// TIA Portal V19 export
FUNCTION "MGF AUTO" : Void   // FC10, LAD
{ S7_Optimized_Access := 'TRUE' }
// stored: SetENOAutomatically false
BEGIN

REGION Network 1
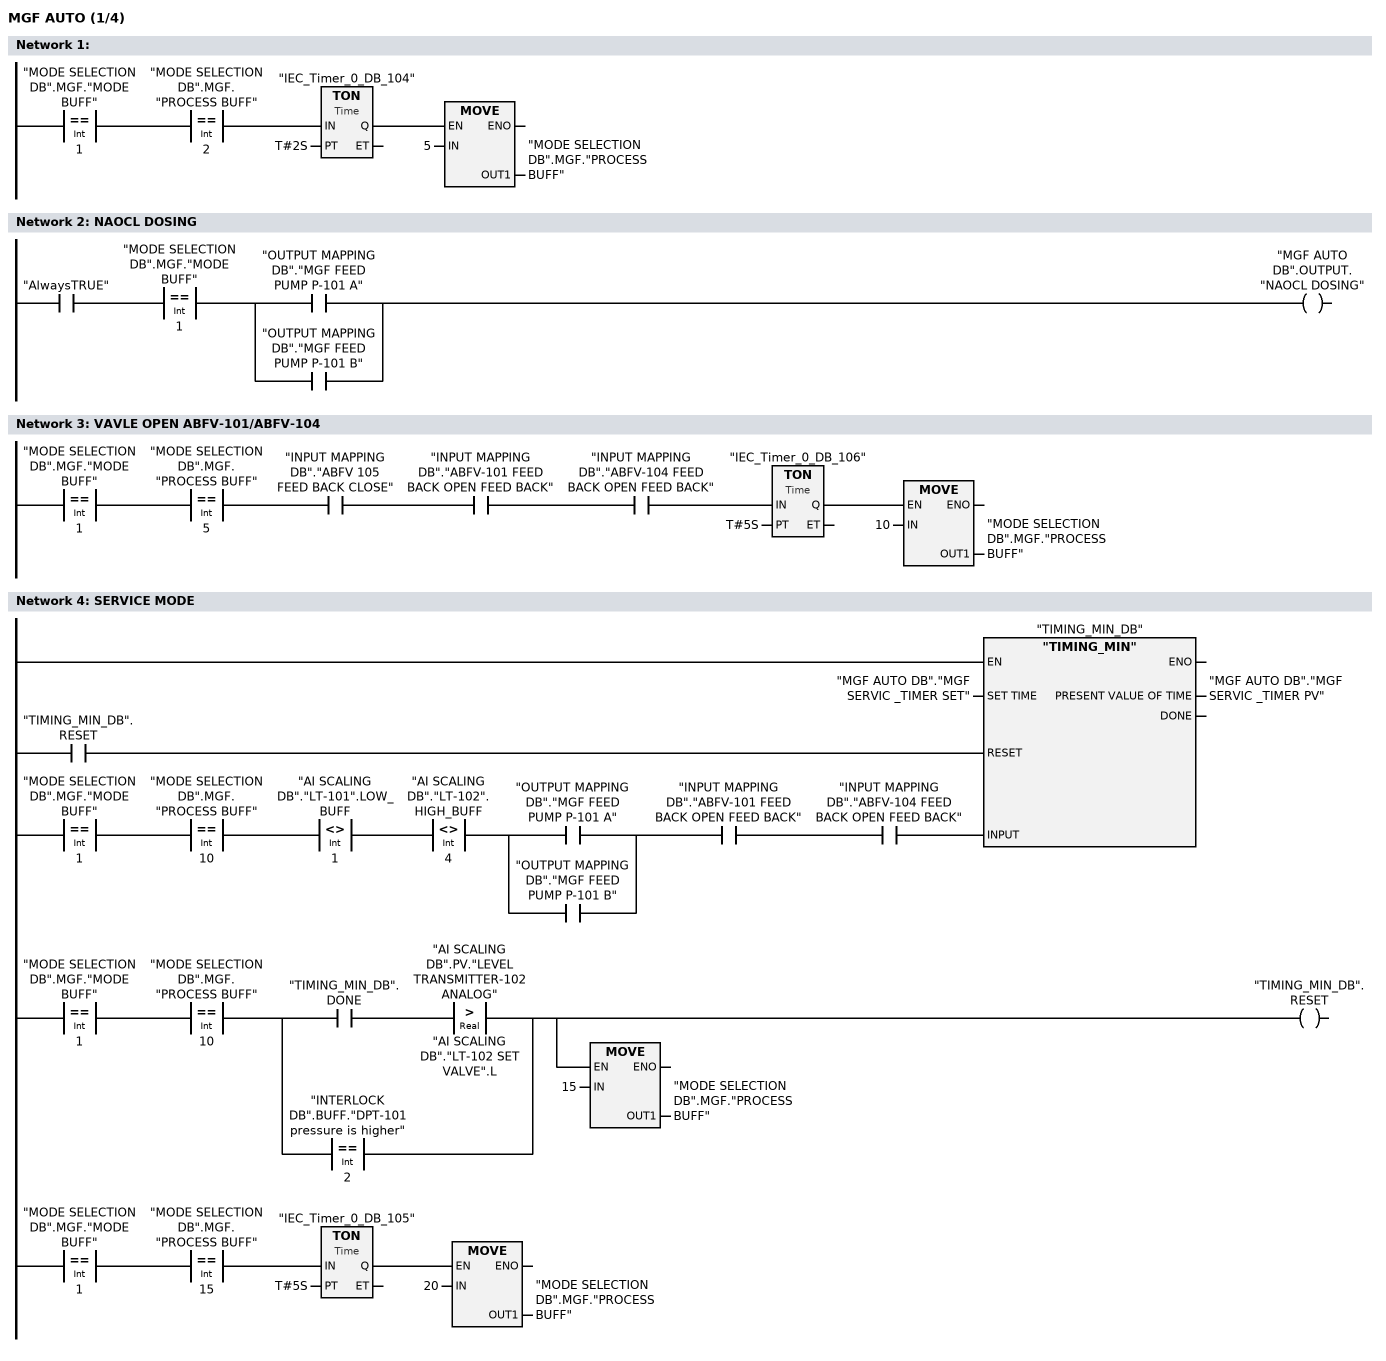
   RUNG wire#powerrail
      { S7_Templates := "SrcType := Int" } EQ_Contact(in1 := "MODE SELECTION DB".MGF."MODE BUFF", in2 := 1)
      { S7_Templates := "SrcType := Int" } EQ_Contact(in1 := "MODE SELECTION DB".MGF."PROCESS BUFF", in2 := 2)
      { S7_Templates := "time_type := Time" } "IEC_Timer_0_DB_104".TON(pt := T#2S, et =>)
      Move(in := 5, out1 => "MODE SELECTION DB".MGF."PROCESS BUFF")
   END_RUNG
   // the same network as SCL:
   "IEC_Timer_0_DB_104".TON(IN := ("MODE SELECTION DB".MGF."MODE BUFF" = 1) AND ("MODE SELECTION DB".MGF."PROCESS BUFF" = 2),
                           PT := T#2S);
   IF "IEC_Timer_0_DB_104".Q THEN "MODE SELECTION DB".MGF."PROCESS BUFF" := 5; END_IF;
END_REGION

REGION Network 2: NAOCL DOSING
   RUNG wire#powerrail
      Contact( "AlwaysTRUE" )
      { S7_Templates := "SrcType := Int" } EQ_Contact(in1 := "MODE SELECTION DB".MGF."MODE BUFF", in2 := 1)
      wire#w1
      Contact( "OUTPUT MAPPING DB"."MGF FEED PUMP P-101 A" )
      wire#w2
      Coil( "MGF AUTO DB".OUTPUT."NAOCL DOSING" )
   END_RUNG
   RUNG wire#w1
      Contact( "OUTPUT MAPPING DB"."MGF FEED PUMP P-101 B" )
   END_RUNG wire#w2
   // the same network as SCL:
   "MGF AUTO DB".OUTPUT."NAOCL DOSING" := "AlwaysTRUE" AND ("MODE SELECTION DB".MGF."MODE BUFF" = 1) AND ("OUTPUT MAPPING DB"."MGF FEED PUMP P-101 A" OR "OUTPUT MAPPING DB"."MGF FEED PUMP P-101 B");
END_REGION

REGION Network 3: VAVLE OPEN ABFV-101/ABFV-104
   RUNG wire#powerrail
      { S7_Templates := "SrcType := Int" } EQ_Contact(in1 := "MODE SELECTION DB".MGF."MODE BUFF", in2 := 1)
      { S7_Templates := "SrcType := Int" } EQ_Contact(in1 := "MODE SELECTION DB".MGF."PROCESS BUFF", in2 := 5)
      Contact( "INPUT MAPPING DB"."ABFV 105 FEED BACK CLOSE" )
      Contact( "INPUT MAPPING DB"."ABFV-101 FEED BACK OPEN FEED BACK" )
      Contact( "INPUT MAPPING DB"."ABFV-104 FEED BACK OPEN FEED BACK" )
      { S7_Templates := "time_type := Time" } "IEC_Timer_0_DB_106".TON(pt := T#5S, et =>)
      Move(in := 10, out1 => "MODE SELECTION DB".MGF."PROCESS BUFF")
   END_RUNG
   // the same network as SCL:
   "IEC_Timer_0_DB_106".TON(IN := ("MODE SELECTION DB".MGF."MODE BUFF" = 1) AND ("MODE SELECTION DB".MGF."PROCESS BUFF" = 5) AND "INPUT MAPPING DB"."ABFV 105 FEED BACK CLOSE" AND "INPUT MAPPING DB"."ABFV-101 FEED BACK OPEN FEED BACK" AND "INPUT MAPPING DB"."ABFV-104 FEED BACK OPEN FEED BACK",
                           PT := T#5S);
   IF "IEC_Timer_0_DB_106".Q THEN "MODE SELECTION DB".MGF."PROCESS BUFF" := 10; END_IF;
END_REGION

REGION Network 4: SERVICE MODE
   RUNG wire#powerrail
      "TIMING_MIN_DB"(RESET := wire#w1, INPUT := wire#w4, "SET TIME" := "MGF AUTO DB"."MGF SERVIC _TIMER SET", "PRESENT VALUE OF TIME" => "MGF AUTO DB"."MGF SERVIC _TIMER PV", DONE =>)
   END_RUNG
   RUNG wire#powerrail
      Contact( "TIMING_MIN_DB".RESET )
   END_RUNG wire#w1
   RUNG wire#powerrail
      { S7_Templates := "SrcType := Int" } EQ_Contact(in1 := "MODE SELECTION DB".MGF."MODE BUFF", in2 := 1)
      { S7_Templates := "SrcType := Int" } EQ_Contact(in1 := "MODE SELECTION DB".MGF."PROCESS BUFF", in2 := 10)
      { S7_Templates := "SrcType := Int" } NE_Contact(in1 := "AI SCALING DB"."LT-101".LOW_BUFF, in2 := 1)
      { S7_Templates := "SrcType := Int" } NE_Contact(in1 := "AI SCALING DB"."LT-102".HIGH_BUFF, in2 := 4)
      wire#w2
      Contact( "OUTPUT MAPPING DB"."MGF FEED PUMP P-101 A" )
      wire#w3
      Contact( "INPUT MAPPING DB"."ABFV-101 FEED BACK OPEN FEED BACK" )
      Contact( "INPUT MAPPING DB"."ABFV-104 FEED BACK OPEN FEED BACK" )
   END_RUNG wire#w4
   RUNG wire#w2
      Contact( "OUTPUT MAPPING DB"."MGF FEED PUMP P-101 B" )
   END_RUNG wire#w3
   RUNG wire#powerrail
      { S7_Templates := "SrcType := Int" } EQ_Contact(in1 := "MODE SELECTION DB".MGF."MODE BUFF", in2 := 1)
      { S7_Templates := "SrcType := Int" } EQ_Contact(in1 := "MODE SELECTION DB".MGF."PROCESS BUFF", in2 := 10)
      wire#w5
      Contact( "TIMING_MIN_DB".DONE )
      { S7_Templates := "SrcType := Real" } GT_Contact(in1 := "AI SCALING DB".PV."LEVEL TRANSMITTER-102 ANALOG", in2 := "AI SCALING DB"."LT-102 SET VALVE".L)
      wire#w6
      Coil( "TIMING_MIN_DB".RESET )
   END_RUNG
   RUNG wire#w5
      { S7_Templates := "SrcType := Int" } EQ_Contact(in1 := "INTERLOCK DB".BUFF."DPT-101 pressure is higher", in2 := 2)
   END_RUNG wire#w6
   RUNG wire#w6
      Move(in := 15, out1 => "MODE SELECTION DB".MGF."PROCESS BUFF")
   END_RUNG
   RUNG wire#powerrail
      { S7_Templates := "SrcType := Int" } EQ_Contact(in1 := "MODE SELECTION DB".MGF."MODE BUFF", in2 := 1)
      { S7_Templates := "SrcType := Int" } EQ_Contact(in1 := "MODE SELECTION DB".MGF."PROCESS BUFF", in2 := 15)
      { S7_Templates := "time_type := Time" } "IEC_Timer_0_DB_105".TON(pt := T#5S, et =>)
      Move(in := 20, out1 => "MODE SELECTION DB".MGF."PROCESS BUFF")
   END_RUNG
   // the same network as SCL:
   "TIMING_MIN_DB"("SET TIME" := "MGF AUTO DB"."MGF SERVIC _TIMER SET",   // "TIMING_MIN"
                   RESET := "TIMING_MIN_DB".RESET,
                   INPUT := ("MODE SELECTION DB".MGF."MODE BUFF" = 1) AND ("MODE SELECTION DB".MGF."PROCESS BUFF" = 10) AND ("AI SCALING DB"."LT-101".LOW_BUFF <> 1) AND ("AI SCALING DB"."LT-102".HIGH_BUFF <> 4) AND ("OUTPUT MAPPING DB"."MGF FEED PUMP P-101 A" OR "OUTPUT MAPPING DB"."MGF FEED PUMP P-101 B") AND "INPUT MAPPING DB"."ABFV-101 FEED BACK OPEN FEED BACK" AND "INPUT MAPPING DB"."ABFV-104 FEED BACK OPEN FEED BACK",
                   "PRESENT VALUE OF TIME" => "MGF AUTO DB"."MGF SERVIC _TIMER PV");
   "TIMING_MIN_DB".RESET := ("MODE SELECTION DB".MGF."MODE BUFF" = 1) AND ("MODE SELECTION DB".MGF."PROCESS BUFF" = 10) AND (("TIMING_MIN_DB".DONE AND ("AI SCALING DB".PV."LEVEL TRANSMITTER-102 ANALOG" > "AI SCALING DB"."LT-102 SET VALVE".L)) OR ("INTERLOCK DB".BUFF."DPT-101 pressure is higher" = 2));
   IF "TIMING_MIN_DB".RESET THEN "MODE SELECTION DB".MGF."PROCESS BUFF" := 15; END_IF;
   "IEC_Timer_0_DB_105".TON(IN := ("MODE SELECTION DB".MGF."MODE BUFF" = 1) AND ("MODE SELECTION DB".MGF."PROCESS BUFF" = 15),
                           PT := T#5S);
   IF "IEC_Timer_0_DB_105".Q THEN "MODE SELECTION DB".MGF."PROCESS BUFF" := 20; END_IF;
END_REGION

REGION Network 5: VAVLE CLOSE ABFV-101/ABFV-104
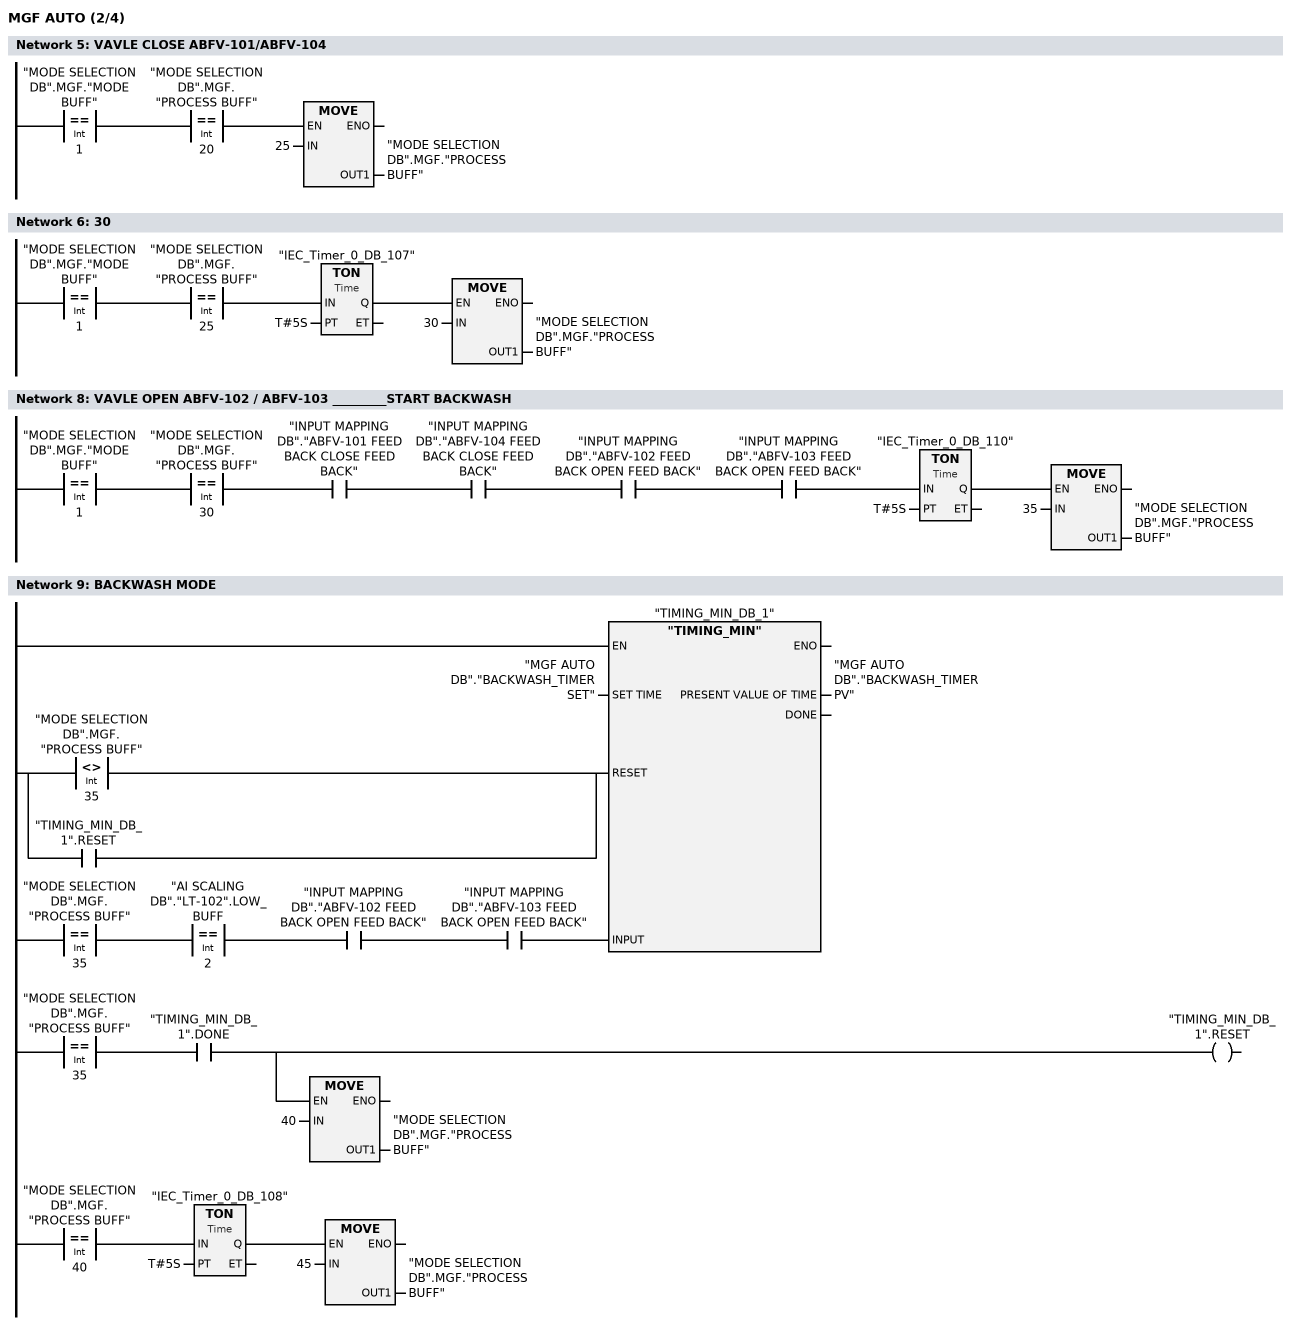
   RUNG wire#powerrail
      { S7_Templates := "SrcType := Int" } EQ_Contact(in1 := "MODE SELECTION DB".MGF."MODE BUFF", in2 := 1)
      { S7_Templates := "SrcType := Int" } EQ_Contact(in1 := "MODE SELECTION DB".MGF."PROCESS BUFF", in2 := 20)
      Move(in := 25, out1 => "MODE SELECTION DB".MGF."PROCESS BUFF")
   END_RUNG
   // the same network as SCL:
   IF ("MODE SELECTION DB".MGF."MODE BUFF" = 1) AND ("MODE SELECTION DB".MGF."PROCESS BUFF" = 20) THEN
       "MODE SELECTION DB".MGF."PROCESS BUFF" := 25;
   END_IF;
END_REGION

REGION Network 6: 30
   RUNG wire#powerrail
      { S7_Templates := "SrcType := Int" } EQ_Contact(in1 := "MODE SELECTION DB".MGF."MODE BUFF", in2 := 1)
      { S7_Templates := "SrcType := Int" } EQ_Contact(in1 := "MODE SELECTION DB".MGF."PROCESS BUFF", in2 := 25)
      { S7_Templates := "time_type := Time" } "IEC_Timer_0_DB_107".TON(pt := T#5S, et =>)
      Move(in := 30, out1 => "MODE SELECTION DB".MGF."PROCESS BUFF")
   END_RUNG
   // the same network as SCL:
   "IEC_Timer_0_DB_107".TON(IN := ("MODE SELECTION DB".MGF."MODE BUFF" = 1) AND ("MODE SELECTION DB".MGF."PROCESS BUFF" = 25),
                           PT := T#5S);
   IF "IEC_Timer_0_DB_107".Q THEN "MODE SELECTION DB".MGF."PROCESS BUFF" := 30; END_IF;
END_REGION

REGION Network 8: VAVLE OPEN ABFV-102 / ABFV-103 _________START BACKWASH
   RUNG wire#powerrail
      { S7_Templates := "SrcType := Int" } EQ_Contact(in1 := "MODE SELECTION DB".MGF."MODE BUFF", in2 := 1)
      { S7_Templates := "SrcType := Int" } EQ_Contact(in1 := "MODE SELECTION DB".MGF."PROCESS BUFF", in2 := 30)
      Contact( "INPUT MAPPING DB"."ABFV-101 FEED BACK CLOSE FEED BACK" )
      Contact( "INPUT MAPPING DB"."ABFV-104 FEED BACK CLOSE FEED BACK" )
      Contact( "INPUT MAPPING DB"."ABFV-102 FEED BACK OPEN FEED BACK" )
      Contact( "INPUT MAPPING DB"."ABFV-103 FEED BACK OPEN FEED BACK" )
      { S7_Templates := "time_type := Time" } "IEC_Timer_0_DB_110".TON(pt := T#5S, et =>)
      Move(in := 35, out1 => "MODE SELECTION DB".MGF."PROCESS BUFF")
   END_RUNG
   // the same network as SCL:
   "IEC_Timer_0_DB_110".TON(IN := ("MODE SELECTION DB".MGF."MODE BUFF" = 1) AND ("MODE SELECTION DB".MGF."PROCESS BUFF" = 30) AND "INPUT MAPPING DB"."ABFV-101 FEED BACK CLOSE FEED BACK" AND "INPUT MAPPING DB"."ABFV-104 FEED BACK CLOSE FEED BACK" AND "INPUT MAPPING DB"."ABFV-102 FEED BACK OPEN FEED BACK" AND "INPUT MAPPING DB"."ABFV-103 FEED BACK OPEN FEED BACK",
                           PT := T#5S);
   IF "IEC_Timer_0_DB_110".Q THEN "MODE SELECTION DB".MGF."PROCESS BUFF" := 35; END_IF;
END_REGION

REGION Network 9: BACKWASH MODE
   RUNG wire#powerrail
      "TIMING_MIN_DB_1"(RESET := wire#w1, INPUT := wire#w2, "SET TIME" := "MGF AUTO DB"."BACKWASH_TIMER SET", "PRESENT VALUE OF TIME" => "MGF AUTO DB"."BACKWASH_TIMER PV", DONE =>)
   END_RUNG
   RUNG wire#powerrail
      { S7_Templates := "SrcType := Int" } NE_Contact(in1 := "MODE SELECTION DB".MGF."PROCESS BUFF", in2 := 35)
   END_RUNG wire#w1
   RUNG wire#powerrail
      Contact( "TIMING_MIN_DB_1".RESET )
   END_RUNG wire#w1
   RUNG wire#powerrail
      { S7_Templates := "SrcType := Int" } EQ_Contact(in1 := "MODE SELECTION DB".MGF."PROCESS BUFF", in2 := 35)
      { S7_Templates := "SrcType := Int" } EQ_Contact(in1 := "AI SCALING DB"."LT-102".LOW_BUFF, in2 := 2)
      Contact( "INPUT MAPPING DB"."ABFV-102 FEED BACK OPEN FEED BACK" )
      Contact( "INPUT MAPPING DB"."ABFV-103 FEED BACK OPEN FEED BACK" )
   END_RUNG wire#w2
   RUNG wire#powerrail
      { S7_Templates := "SrcType := Int" } EQ_Contact(in1 := "MODE SELECTION DB".MGF."PROCESS BUFF", in2 := 35)
      Contact( "TIMING_MIN_DB_1".DONE )
      wire#w3
      Coil( "TIMING_MIN_DB_1".RESET )
   END_RUNG
   RUNG wire#w3
      Move(in := 40, out1 => "MODE SELECTION DB".MGF."PROCESS BUFF")
   END_RUNG
   RUNG wire#powerrail
      { S7_Templates := "SrcType := Int" } EQ_Contact(in1 := "MODE SELECTION DB".MGF."PROCESS BUFF", in2 := 40)
      { S7_Templates := "time_type := Time" } "IEC_Timer_0_DB_108".TON(pt := T#5S, et =>)
      Move(in := 45, out1 => "MODE SELECTION DB".MGF."PROCESS BUFF")
   END_RUNG
   // the same network as SCL:
   "TIMING_MIN_DB_1"("SET TIME" := "MGF AUTO DB"."BACKWASH_TIMER SET",   // "TIMING_MIN"
                     RESET := ("MODE SELECTION DB".MGF."PROCESS BUFF" <> 35) OR "TIMING_MIN_DB_1".RESET,
                     INPUT := ("MODE SELECTION DB".MGF."PROCESS BUFF" = 35) AND ("AI SCALING DB"."LT-102".LOW_BUFF = 2) AND "INPUT MAPPING DB"."ABFV-102 FEED BACK OPEN FEED BACK" AND "INPUT MAPPING DB"."ABFV-103 FEED BACK OPEN FEED BACK",
                     "PRESENT VALUE OF TIME" => "MGF AUTO DB"."BACKWASH_TIMER PV");
   "TIMING_MIN_DB_1".RESET := ("MODE SELECTION DB".MGF."PROCESS BUFF" = 35) AND "TIMING_MIN_DB_1".DONE;
   IF "TIMING_MIN_DB_1".RESET THEN "MODE SELECTION DB".MGF."PROCESS BUFF" := 40; END_IF;
   "IEC_Timer_0_DB_108".TON(IN := "MODE SELECTION DB".MGF."PROCESS BUFF" = 40, PT := T#5S);
   IF "IEC_Timer_0_DB_108".Q THEN "MODE SELECTION DB".MGF."PROCESS BUFF" := 45; END_IF;
END_REGION

REGION Network 10: VALVE CLOSE
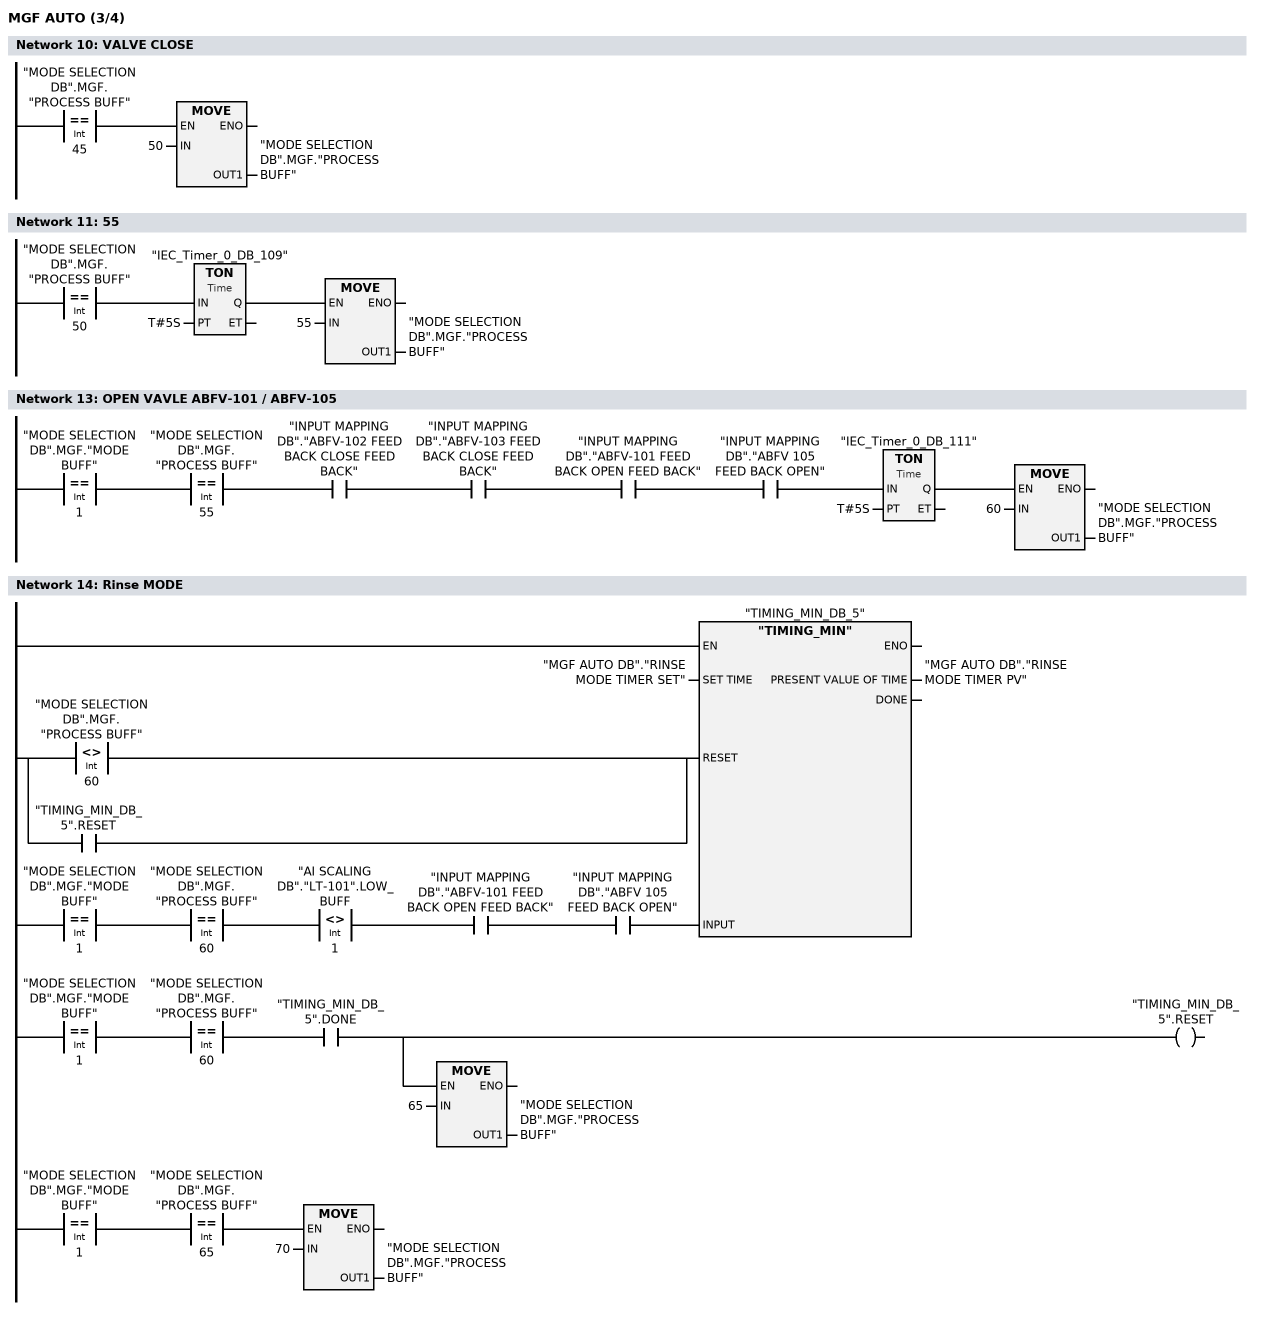
   RUNG wire#powerrail
      { S7_Templates := "SrcType := Int" } EQ_Contact(in1 := "MODE SELECTION DB".MGF."PROCESS BUFF", in2 := 45)
      Move(in := 50, out1 => "MODE SELECTION DB".MGF."PROCESS BUFF")
   END_RUNG
   // the same network as SCL:
   IF "MODE SELECTION DB".MGF."PROCESS BUFF" = 45 THEN "MODE SELECTION DB".MGF."PROCESS BUFF" := 50; END_IF;
END_REGION

REGION Network 11: 55
   RUNG wire#powerrail
      { S7_Templates := "SrcType := Int" } EQ_Contact(in1 := "MODE SELECTION DB".MGF."PROCESS BUFF", in2 := 50)
      { S7_Templates := "time_type := Time" } "IEC_Timer_0_DB_109".TON(pt := T#5S, et =>)
      Move(in := 55, out1 => "MODE SELECTION DB".MGF."PROCESS BUFF")
   END_RUNG
   // the same network as SCL:
   "IEC_Timer_0_DB_109".TON(IN := "MODE SELECTION DB".MGF."PROCESS BUFF" = 50, PT := T#5S);
   IF "IEC_Timer_0_DB_109".Q THEN "MODE SELECTION DB".MGF."PROCESS BUFF" := 55; END_IF;
END_REGION

REGION Network 13: OPEN VAVLE ABFV-101 / ABFV-105
   RUNG wire#powerrail
      { S7_Templates := "SrcType := Int" } EQ_Contact(in1 := "MODE SELECTION DB".MGF."MODE BUFF", in2 := 1)
      { S7_Templates := "SrcType := Int" } EQ_Contact(in1 := "MODE SELECTION DB".MGF."PROCESS BUFF", in2 := 55)
      Contact( "INPUT MAPPING DB"."ABFV-102 FEED BACK CLOSE FEED BACK" )
      Contact( "INPUT MAPPING DB"."ABFV-103 FEED BACK CLOSE FEED BACK" )
      Contact( "INPUT MAPPING DB"."ABFV-101 FEED BACK OPEN FEED BACK" )
      Contact( "INPUT MAPPING DB"."ABFV 105 FEED BACK OPEN" )
      { S7_Templates := "time_type := Time" } "IEC_Timer_0_DB_111".TON(pt := T#5S, et =>)
      Move(in := 60, out1 => "MODE SELECTION DB".MGF."PROCESS BUFF")
   END_RUNG
   // the same network as SCL:
   "IEC_Timer_0_DB_111".TON(IN := ("MODE SELECTION DB".MGF."MODE BUFF" = 1) AND ("MODE SELECTION DB".MGF."PROCESS BUFF" = 55) AND "INPUT MAPPING DB"."ABFV-102 FEED BACK CLOSE FEED BACK" AND "INPUT MAPPING DB"."ABFV-103 FEED BACK CLOSE FEED BACK" AND "INPUT MAPPING DB"."ABFV-101 FEED BACK OPEN FEED BACK" AND "INPUT MAPPING DB"."ABFV 105 FEED BACK OPEN",
                           PT := T#5S);
   IF "IEC_Timer_0_DB_111".Q THEN "MODE SELECTION DB".MGF."PROCESS BUFF" := 60; END_IF;
END_REGION

REGION Network 14: Rinse MODE
   RUNG wire#powerrail
      "TIMING_MIN_DB_5"(RESET := wire#w1, INPUT := wire#w2, "SET TIME" := "MGF AUTO DB"."RINSE MODE TIMER SET", "PRESENT VALUE OF TIME" => "MGF AUTO DB"."RINSE MODE TIMER PV", DONE =>)
   END_RUNG
   RUNG wire#powerrail
      { S7_Templates := "SrcType := Int" } NE_Contact(in1 := "MODE SELECTION DB".MGF."PROCESS BUFF", in2 := 60)
   END_RUNG wire#w1
   RUNG wire#powerrail
      Contact( "TIMING_MIN_DB_5".RESET )
   END_RUNG wire#w1
   RUNG wire#powerrail
      { S7_Templates := "SrcType := Int" } EQ_Contact(in1 := "MODE SELECTION DB".MGF."MODE BUFF", in2 := 1)
      { S7_Templates := "SrcType := Int" } EQ_Contact(in1 := "MODE SELECTION DB".MGF."PROCESS BUFF", in2 := 60)
      { S7_Templates := "SrcType := Int" } NE_Contact(in1 := "AI SCALING DB"."LT-101".LOW_BUFF, in2 := 1)
      Contact( "INPUT MAPPING DB"."ABFV-101 FEED BACK OPEN FEED BACK" )
      Contact( "INPUT MAPPING DB"."ABFV 105 FEED BACK OPEN" )
   END_RUNG wire#w2
   RUNG wire#powerrail
      { S7_Templates := "SrcType := Int" } EQ_Contact(in1 := "MODE SELECTION DB".MGF."MODE BUFF", in2 := 1)
      { S7_Templates := "SrcType := Int" } EQ_Contact(in1 := "MODE SELECTION DB".MGF."PROCESS BUFF", in2 := 60)
      Contact( "TIMING_MIN_DB_5".DONE )
      wire#w3
      Coil( "TIMING_MIN_DB_5".RESET )
   END_RUNG
   RUNG wire#w3
      Move(in := 65, out1 => "MODE SELECTION DB".MGF."PROCESS BUFF")
   END_RUNG
   RUNG wire#powerrail
      { S7_Templates := "SrcType := Int" } EQ_Contact(in1 := "MODE SELECTION DB".MGF."MODE BUFF", in2 := 1)
      { S7_Templates := "SrcType := Int" } EQ_Contact(in1 := "MODE SELECTION DB".MGF."PROCESS BUFF", in2 := 65)
      Move(in := 70, out1 => "MODE SELECTION DB".MGF."PROCESS BUFF")
   END_RUNG
   // the same network as SCL:
   "TIMING_MIN_DB_5"("SET TIME" := "MGF AUTO DB"."RINSE MODE TIMER SET",   // "TIMING_MIN"
                     RESET := ("MODE SELECTION DB".MGF."PROCESS BUFF" <> 60) OR "TIMING_MIN_DB_5".RESET,
                     INPUT := ("MODE SELECTION DB".MGF."MODE BUFF" = 1) AND ("MODE SELECTION DB".MGF."PROCESS BUFF" = 60) AND ("AI SCALING DB"."LT-101".LOW_BUFF <> 1) AND "INPUT MAPPING DB"."ABFV-101 FEED BACK OPEN FEED BACK" AND "INPUT MAPPING DB"."ABFV 105 FEED BACK OPEN",
                     "PRESENT VALUE OF TIME" => "MGF AUTO DB"."RINSE MODE TIMER PV");
   "TIMING_MIN_DB_5".RESET := ("MODE SELECTION DB".MGF."MODE BUFF" = 1) AND ("MODE SELECTION DB".MGF."PROCESS BUFF" = 60) AND "TIMING_MIN_DB_5".DONE;
   IF "TIMING_MIN_DB_5".RESET THEN "MODE SELECTION DB".MGF."PROCESS BUFF" := 65; END_IF;
   IF ("MODE SELECTION DB".MGF."MODE BUFF" = 1) AND ("MODE SELECTION DB".MGF."PROCESS BUFF" = 65) THEN
       "MODE SELECTION DB".MGF."PROCESS BUFF" := 70;
   END_IF;
END_REGION

REGION Network 15: VALVE CLOSE
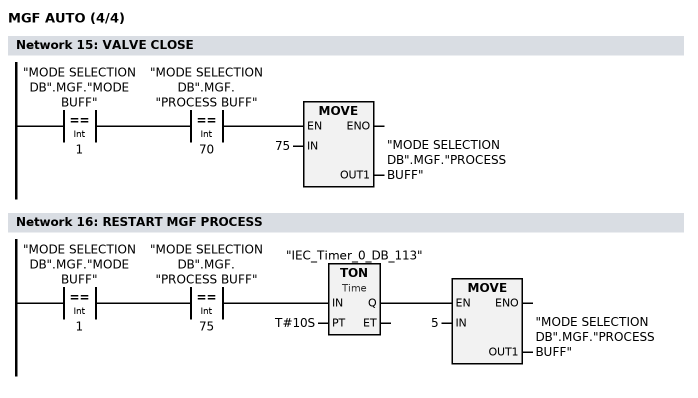
   RUNG wire#powerrail
      { S7_Templates := "SrcType := Int" } EQ_Contact(in1 := "MODE SELECTION DB".MGF."MODE BUFF", in2 := 1)
      { S7_Templates := "SrcType := Int" } EQ_Contact(in1 := "MODE SELECTION DB".MGF."PROCESS BUFF", in2 := 70)
      Move(in := 75, out1 => "MODE SELECTION DB".MGF."PROCESS BUFF")
   END_RUNG
   // the same network as SCL:
   IF ("MODE SELECTION DB".MGF."MODE BUFF" = 1) AND ("MODE SELECTION DB".MGF."PROCESS BUFF" = 70) THEN
       "MODE SELECTION DB".MGF."PROCESS BUFF" := 75;
   END_IF;
END_REGION

REGION Network 16: RESTART MGF PROCESS
   RUNG wire#powerrail
      { S7_Templates := "SrcType := Int" } EQ_Contact(in1 := "MODE SELECTION DB".MGF."MODE BUFF", in2 := 1)
      { S7_Templates := "SrcType := Int" } EQ_Contact(in1 := "MODE SELECTION DB".MGF."PROCESS BUFF", in2 := 75)
      { S7_Templates := "time_type := Time" } "IEC_Timer_0_DB_113".TON(pt := T#10S, et =>)
      Move(in := 5, out1 => "MODE SELECTION DB".MGF."PROCESS BUFF")
   END_RUNG
   // the same network as SCL:
   "IEC_Timer_0_DB_113".TON(IN := ("MODE SELECTION DB".MGF."MODE BUFF" = 1) AND ("MODE SELECTION DB".MGF."PROCESS BUFF" = 75),
                           PT := T#10S);
   IF "IEC_Timer_0_DB_113".Q THEN "MODE SELECTION DB".MGF."PROCESS BUFF" := 5; END_IF;
END_REGION
END_FUNCTION
